(* IEC 61131-3 sources: Lasal/CPU_5344_V01/Class/ctrlLubricate, 1 file *)

(* ---- ctrlLubricate.st ---- *)
(*!
<Class
	Name               = "ctrlLubricate"
	Revision           = "0.0"
	RealtimeTask       = "false"
	CyclicTask         = "true"
	DefCyclictime      = "10 ms"
	BackgroundTask     = "false"
	Sigmatek           = "false"
	OSInterface        = "false"
	HighPriority       = "false"
	Automatic          = "false"
	UpdateMode         = "Prescan"
	SharedCommandTable = "true"
	Objectsize         = "(540,480)">
	<Channels>
		<Server Name="Actuate" Visualized="true" Initialize="false" WriteProtected="false" Retentive="false"/>
		<Server Name="ClassSvr" Visualized="false" Initialize="false" WriteProtected="true" Retentive="false"/>
		<Server Name="CycleTIme" Visualized="false" Initialize="false" WriteProtected="true" Retentive="false"/>
		<Server Name="Offtime" Visualized="true" Initialize="true" DefValue="400" WriteProtected="false" Retentive="File"/>
		<Server Name="Ontime" Visualized="true" Initialize="true" DefValue="200" WriteProtected="false" Retentive="File"/>
		<Server Name="Stepper" Visualized="false" Initialize="false" WriteProtected="true" Retentive="false"/>
		<Server Name="TotalCycleTime" Visualized="false" Initialize="false" WriteProtected="true" Retentive="false"/>
		<Client Name="Air" Required="false" Internal="false"/>
		<Client Name="iEnableLubricate" Required="false" Internal="false"/>
		<Client Name="iPulsesPerSecond" Required="true" Internal="false"/>
		<Client Name="Oil" Required="false" Internal="false"/>
	</Channels>
</Class>
*)
ctrlLubricate : CLASS
  //Servers:
	ClassSvr 	: SvrChCmd_DINT;
	Stepper 	: SvrCh_DINT;
	CycleTIme 	: SvrCh_UDINT;
	TotalCycleTime 	: SvrCh_UDINT;
	Ontime 	: SvrCh_UDINT;
	Offtime 	: SvrCh_UDINT;
	Actuate 	: SvrCh_DINT;
  //Clients:
	Oil 	: CltCh_DINT;
	Air 	: CltCh_DINT;
	iPulsesPerSecond 	: CltCh_DINT;
	iEnableLubricate 	: CltCh_DINT;
  //Variables:
  //Functions:

	FUNCTION VIRTUAL GLOBAL CyWork
		VAR_INPUT
			EAX 	: UDINT;
		END_VAR
		VAR_OUTPUT
			state (EAX) 	: UDINT;
		END_VAR;

	FUNCTION GLOBAL Smeren;

	FUNCTION ReadInputs;

	FUNCTION WriteOutputs;

	FUNCTION GLOBAL Start;

	FUNCTION GLOBAL Stop;
  //Tables:
	FUNCTION @STD
		VAR_OUTPUT
			ret_code	: CONFSTATES;
		END_VAR;
	FUNCTION GLOBAL TAB @CT_;
END_CLASS;

// JdK 7-8-2019 ctrlLubricate copied from 4090 to 4284
// function is to control lubrication with oil and sometimes air, if no air offtime will be 0, so oil is continue on

FUNCTION VIRTUAL GLOBAL ctrlLubricate::CyWork
	VAR_INPUT
		EAX 	: UDINT;
	END_VAR
	VAR_OUTPUT
		state (EAX) 	: UDINT;
	END_VAR

  ReadInputs();

  if Actuate | iEnableLubricate then // als het object smering aangeroepen wordt wordt de functie gestart
    Smeren();
  else // als het startsignaal niet aanwezig is of afvalt dan worden de startcondities gezet
    Stepper := 0;
    Air := FALSE;
    Oil := FALSE;
  end_if;

  WriteOutputs();

	state := READY;

END_FUNCTION

FUNCTION GLOBAL ctrlLubricate::Smeren

  TotalCycleTime := Ontime + Offtime; // berekenen van de totale cycletijd nav de inputvariabelen

  case Stepper of

  0: //  starttijd van de cyclus vasststellen en lucht en olie inschakelen
    CycleTime := ops.tAbsolute;
    Air := TRUE;
    Oil := TRUE;
    if Offtime > 0 then //else just keep everything on
      Stepper +=1;
    end_if;

  1:// Olie uitschakelen als ontime verstreken is
    if ops.tAbsolute - CycleTime > Ontime then
      Oil := FALSE;
      Stepper +=1;
    end_if;

  2: // weer terug naar begin en dus olie weer inschakelen na verstrijken van totale cycletijd
    if ops.tAbsolute - CycleTime > TotalCycleTime then
      Stepper := 0;
    end_if;

  end_case;

END_FUNCTION

FUNCTION ctrlLubricate::ReadInputs
iPulsesPerSecond := iPulsesPerSecond.Read();
iEnableLubricate := iEnableLubricate.Read();

if iPulsesPerSecond > 0 then
  Offtime := 60000 / to_udint(iPulsesPerSecond);
end_if;

END_FUNCTION

FUNCTION ctrlLubricate::WriteOutputs

  Air.Write(Air);
  Oil.Write(Oil);

END_FUNCTION

FUNCTION GLOBAL ctrlLubricate::Start

  Actuate := TRUE;

END_FUNCTION

FUNCTION GLOBAL ctrlLubricate::Stop

  Actuate := FALSE;

END_FUNCTION
